PROGRAM pouHMI
VAR
END_VAR

//all logic to control HMI
prgHMIcontrol();

//control Unit Screen
prgHMIUnits();

//logic for stations
prgHMIstations();

//call to read text lists into PLC memory arrays
prgReadTextList();

//control language Screen
prgHMILanguage();

//axis telegram diag screen
prgHMIaxis();

//lock station logic
actLockStation();

ACTION actLockStation:
//lock stations together feedback

IF gHMIButtons.btnLockStation1 THEN gHMIData.gStateLockStation1 := 1; ELSE gHMIData.gStateLockStation1 := 0 ; END_IF
IF gHMIButtons.btnLockStation2 THEN gHMIData.gStateLockStation2 := 1; ELSE gHMIData.gStateLockStation2 := 0 ; END_IF
IF gHMIButtons.btnLockStation3 THEN gHMIData.gStateLockStation3 := 1; ELSE gHMIData.gStateLockStation3 := 0 ; END_IF	
IF gHMIButtons.btnLockStation4 THEN gHMIData.gStateLockStation4 := 1; ELSE gHMIData.gStateLockStation4 := 0 ; END_IF
IF gHMIButtons.btnLockStation5 THEN gHMIData.gStateLockStation5 := 1; ELSE gHMIData.gStateLockStation5 := 0 ; END_IF
IF gHMIButtons.btnLockStation6 THEN gHMIData.gStateLockStation6 := 1; ELSE gHMIData.gStateLockStation6 := 0 ; END_IF
END_ACTION

ACTION actResetButtonPress:
//if its on, then turn it off, it will be taken in other places
IF gHMIButtons.gAnyButtonPressed AND System.PulseTenSecond THEN
	gHMIButtons.gAnyButtonPressed := FALSE;
END_IF
END_ACTION

END_PROGRAM

(* stored: Version 1.1.0.1, ProductVersion 3.1.4024.11
   POU pouHMI: Id {54e7270f-e089-40a6-a429-6d01839a041f}, SpecialFunc None
   Action actLockStation: Id {c61404f0-1138-0bfa-3f97-ad7ee6ec469e}
   Action actResetButtonPress: Id {e16beb8b-09dd-0fd9-2961-1cc1cb91a6de} *)
